FUNCTION udfhgdshfksfkjshdkjfdhsfsdfsdfsfsdfsdfsdsdf : sdfdsfsdfsd
VAR_INPUT
END_VAR
VAR
END_VAR

END_FUNCTION

(* stored: Version 1.1.0.1, ProductVersion 3.1.4026.12
   POU udfhgdshfksfkjshdkjfdhsfsdfsdfsfsdfsdfsdsdf: Id {5933dbdd-385d-40f4-9103-aac4038dca7a}, SpecialFunc None *)
